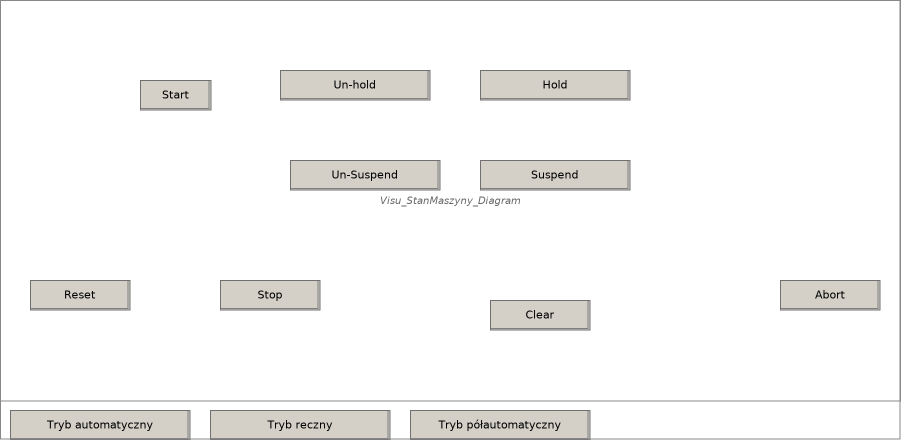
VISUALIZATION Visu_StanMaszyny_DiagramZPrzyciskami  // 901x440
VAR_IN_OUT
	
END_VAR
VAR_INPUT
	bWlaczPrzyciski								: BOOL;
END_VAR
    Frame (0,0 901x401)
        shows Visu_StanMaszyny_Diagram(bWlaczPrzyciski := bWlaczPrzyciski)
    Button (140,80 71x30), "Start", colour toggle: GVL_Elementy.fbPrzysciskStart.bPodswietlenie
        tap GVL_StanMaszyny.bStart
    Button (220,280 100x30), "Stop", colour toggle: GVL_Elementy.fbPrzyciskStop.bPodswietlenie
        tap GVL_StanMaszyny.bStop
    Button (30,280 100x30), "Reset"
        tap GVL_StanMaszyny.bReset
    Button (780,280 100x30), "Abort"
        tap GVL_StanMaszyny.bAbort
    Button (480,70 150x30), "Hold", invisible if: not GVL_StanMaszyny.fbStanMaszyny.arrVisuTryb[GVL_StanMaszyny.fbStanMaszyny.iNumerTrybuPracy][11]
        tap GVL_StanMaszyny.bHold
    Button (280,70 150x30), "Un-hold", invisible if: not GVL_StanMaszyny.fbStanMaszyny.arrVisuTryb[GVL_StanMaszyny.fbStanMaszyny.iNumerTrybuPracy][11]
        tap GVL_StanMaszyny.bUnhold
    Button (480,160 150x30), "Suspend", invisible if: not GVL_StanMaszyny.fbStanMaszyny.arrVisuTryb[GVL_StanMaszyny.fbStanMaszyny.iNumerTrybuPracy][5]
        tap GVL_StanMaszyny.bSuspend
    Button (290,160 150x30), "Un-Suspend", invisible if: not GVL_StanMaszyny.fbStanMaszyny.arrVisuTryb[GVL_StanMaszyny.fbStanMaszyny.iNumerTrybuPracy][5]
        tap GVL_StanMaszyny.bUnsuspend
    Button (10,410 180x30), "Tryb automatyczny", colour toggle: GVL_StanMaszyny.eTrybPracy = E_PMLUnitMode.AUTOMATIC, input disabled if: not (GVL_StanMaszyny.fbStanMaszyny.eStan = E_PMLState.ABORTED or GVL_StanMaszyny.fbStanMaszyny.eStan = E_PMLState.STOPPED)
        OnMouseDown: execute { GVL_StanMaszyny.eTrybPracy	:= E_PMLUnitMode.AUTOMATIC; }
    Button (210,410 180x30), "Tryb reczny", colour toggle: GVL_StanMaszyny.eTrybPracy = E_PMLUnitMode.MANUAL, input disabled if: not (GVL_StanMaszyny.fbStanMaszyny.eStan = E_PMLState.ABORTED or GVL_StanMaszyny.fbStanMaszyny.eStan = E_PMLState.STOPPED)
        OnMouseDown: execute { GVL_StanMaszyny.eTrybPracy	:= E_PMLUnitMode.MANUAL; }
    Button (490,300 100x30), "Clear"
        tap GVL_StanMaszyny.bClear
    Button (410,410 180x30), "Tryb półautomatyczny", colour toggle: GVL_StanMaszyny.eTrybPracy = E_PMLUnitMode.SEMIAUTOMATIC, input disabled if: not (GVL_StanMaszyny.fbStanMaszyny.eStan = E_PMLState.ABORTED or GVL_StanMaszyny.fbStanMaszyny.eStan = E_PMLState.STOPPED)
        OnMouseDown: execute { GVL_StanMaszyny.eTrybPracy	:= E_PMLUnitMode.SEMIAUTOMATIC; }
END_VISUALIZATION

(* stored: Version 1.1.0.1, ProductVersion 3.1.4024.11
   Visu Visu_StanMaszyny_DiagramZPrzyciskami: Id {d394ae5d-88aa-493b-b8e4-1e05743494e2} *)
